FUNCTION_BLOCK DiaglogsContext EXTENDS TcoCore.TcoContext
VAR
    _invokeDiaglog1 : BOOL;
    _dialog1        : TcoCore.TcoDialog(THIS^);
    _dialog2        : TcoCore.TcoDialog(THIS^);
    _dialog3        : TcoCore.TcoDialog(THIS^);
	_dialog4        : TcoCore.TcoDialog(THIS^);

    _invokeDiaglogsConsequential : BOOL;
    _dialog1Consequential        : TcoCore.TcoDialog(THIS^);
    _dialog2Consequential        : TcoCore.TcoDialog(THIS^);
    _dialog3Consequential        : TcoCore.TcoDialog(THIS^);
	
	diag: ITcoDialogAnswer;
	_tonDisposeDialog: TON;
    _state : INT;
	
	
    _invokeCustomizedDiaglog : BOOL;
    _dialogCustomized        : TcoCore.TcoCustomizedDialog(THIS^);
    
END_VAR

(*~
	<docu>
		<summary>
			Main method of the TcoContext. This is the entry point of any control logic that belongs to this context. 
			The call of this method is ensured by calling the <c>InstanceName.Run()</c> method, and it must not be called explicitly.
			This method is abstract, and it must be overridden in derived block.
		</summary>
	</docu>
~*)
METHOD PROTECTED  Main
VAR

END_VAR

CASE _state OF
    0:
        IF (_invokeDiaglog1) THEN
            _state := 10;
		ELSIF (_invokeCustomizedDiaglog) THEN
            _state := 50;
        
        END_IF;
    10:
        _dialog1.Show()
            .WithType(eDialogType.Question)
            .WithYesNoCancel()
			.WithImage('D:\MTS\Develop\TcOpenGroup\TcOpen\assets\logo\TcOpenLogo.png',500,500)
            .WithCaption('Hey 1')
            .WithText('Do we go ahead to 2?');

        IF (_dialog1.Answer = TcoCore.eDialogAnswer.Yes) THEN
            _state := 15;
        END_IF;

        IF (_dialog1.Answer = TcoCore.eDialogAnswer.No) THEN
            _state := 1000;
        END_IF;

        IF (_dialog1.Answer = TcoCore.eDialogAnswer.Cancel) THEN
            _state := 0;
            _invokeDiaglog1 := FALSE;
        END_IF;
    15:
        _dialog1.Show()
            .WithType(eDialogType.Question)
            .WithYesNoCancel()
			.WithImage('',500,500)
            .WithCaption('Hey 2')
            .WithText('Do we go ahead?');

        IF (_dialog1.Answer = TcoCore.eDialogAnswer.Yes) THEN
            _state := 20;
        END_IF;

        IF (_dialog1.Answer = TcoCore.eDialogAnswer.No) THEN
            _state := 1000;
        END_IF;

        IF (_dialog1.Answer = TcoCore.eDialogAnswer.Cancel) THEN
            _state := 0;
            _invokeDiaglog1 := FALSE;
        END_IF;
    20:
        IF (_dialog2.Show()
            .WithType(eDialogType.Info)
            .WithOk()
            .WithCaption('Hey')
            .WithText('We go ahead.')
            .Answer =
            TcoCore.eDialogAnswer.OK) THEN
            _state := 30;
        END_IF
    30:
        _state := 40;
        _tonDisposeDialog(In := FALSE);
    40:
        _tonDisposeDialog(IN := TRUE, PT := T#4S);
		_dialog4.ShowWithExternalClose(inOkAnswerSignal:=FALSE , inYesAnswerSignal:= _tonDisposeDialog.Q, inNoAnswerSignal:= FALSE, inCancelAnswerSignal:= FALSE)
		    .WithType(eDialogType.Info)
            .WithYesNoCancel()
            .WithCaption('Hey')
            .WithText('Do you wana retry it? Yes answer will be set in 4 sec?');

        IF (_dialog4.Answer = TcoCore.eDialogAnswer.Yes) THEN
            _state := 0;
        END_IF;

        IF (_dialog4.Answer = TcoCore.eDialogAnswer.No) THEN
            _state := 50;
        END_IF;

        IF (_dialog4.Answer = TcoCore.eDialogAnswer.Cancel) THEN
            _state := 0;
            _invokeDiaglog1 := FALSE;
        END_IF;
	50:
         _dialogCustomized.Show()
            .WithType(eDialogType.Info)
            .WithOption1('This is Option1=>retry')
			  .WithOption2('This is Option2=>first step')
			    .WithOption3('This is Option3 =>continue')
				  .WithOption4('This is Option4=>stop sequence')
            .WithCaption('Hey')
            .WithText('What we are going to do.');
            
			 IF (_dialogCustomized.Answer = TcoCore.eCustomizedDialogAnswer.Option1) THEN
				_state := 50;
			END_IF;
	
			IF (_dialogCustomized.Answer = TcoCore.eCustomizedDialogAnswer.Option2) THEN
				_state := 0;
			END_IF;
	
			IF (_dialogCustomized.Answer = TcoCore.eCustomizedDialogAnswer.Option3) THEN
				_state := 51;
			END_IF;
	
			IF (_dialogCustomized.Answer = TcoCore.eCustomizedDialogAnswer.Option4) THEN
				_state := 0;
				_invokeCustomizedDiaglog := FALSE;
				_invokeDiaglog1 := FALSE;
			END_IF;
	51:
         _dialogCustomized.Show()
            
            .WithOption1('This is Option1=>retry')
			  .WithOption2('This is Option2=>first step')
			    .WithOption3('This is Option3 =>continue')
			.WithImage('D:\MTS\Develop\TcOpenGroup\TcOpen\assets\logo\TcOpenWide.png',500,500)
            .WithCaption('Hey')
            .WithText('What we are going to do.');
            
			 IF (_dialogCustomized.Answer = TcoCore.eCustomizedDialogAnswer.Option1) THEN
				_state := 50;
			END_IF;
	
			IF (_dialogCustomized.Answer = TcoCore.eCustomizedDialogAnswer.Option2) THEN
				_state := 0;
			END_IF;
	
			IF (_dialogCustomized.Answer = TcoCore.eCustomizedDialogAnswer.Option3) THEN
				_state := 60;
			END_IF;
	
			IF (_dialogCustomized.Answer = TcoCore.eCustomizedDialogAnswer.Option4) THEN
				_state := 0;
				_invokeCustomizedDiaglog := FALSE;
				_invokeDiaglog1 := FALSE;
			END_IF;
     
     
    60:
        _state := 70;
        _tonDisposeDialog(In := FALSE);
	70:
        _tonDisposeDialog(IN := TRUE, PT := T#4S);
		_dialog4.ShowWithExternalClose(inOkAnswerSignal:=FALSE , inYesAnswerSignal:= _tonDisposeDialog.Q, inNoAnswerSignal:= FALSE, inCancelAnswerSignal:= FALSE)
		    .WithType(eDialogType.Info)
            .WithYesNoCancel()
            .WithCaption('Hey')
            .WithText('Do you wana retry it? Yes answer will be set in 4 sec?');

        IF (_dialog4.Answer = TcoCore.eDialogAnswer.Yes) THEN
            _state := 0;
        END_IF;

        IF (_dialog4.Answer = TcoCore.eDialogAnswer.No) THEN
            _state := 80;
        END_IF;

        IF (_dialog4.Answer = TcoCore.eDialogAnswer.Cancel) THEN
            _state := 0;
            _invokeDiaglog1 := FALSE;
        END_IF;
		
	 80:
        _state := 90;
        _tonDisposeDialog(In := FALSE);
	90:
        _tonDisposeDialog(IN := TRUE, PT := T#4S);
		 _dialogCustomized.ShowWithExternalClose(inOption1AnswerSignal:=FALSE,inOption2AnswerSignal:=FALSE, inOption3AnswerSignal:=_tonDisposeDialog.Q,inOption4AnswerSignal:=FALSE)
            
            .WithOption1('This is Option1=>retry')
			  .WithOption2('This is Option2=>first step')
			    .WithOption3('This is Option3 =>continue and finish in 4s')
			.WithImage('D:\MTS\Develop\TcOpenGroup\TcOpen\assets\logo\TcOpenWide.png',500,500)
            .WithCaption('Hey')
            .WithText('What we are going to do.');
            
		
            
			 IF (_dialogCustomized.Answer = TcoCore.eCustomizedDialogAnswer.Option1) THEN
				_state := 80;
			END_IF;
	
			IF (_dialogCustomized.Answer = TcoCore.eCustomizedDialogAnswer.Option2) THEN
				_state := 0;
			END_IF;
	
			IF (_dialogCustomized.Answer = TcoCore.eCustomizedDialogAnswer.Option3) THEN
				_state := 0;
				_invokeCustomizedDiaglog := FALSE;
				_invokeDiaglog1 := FALSE;
			END_IF;
		
	
    1000:
        IF (_dialog3.Show()
            .WithType(eDialogType.Warning)
            .WithOk()
            .WithCaption('Hey')
            .WithText('We don`t go ahead.')
            .Answer =
            TcoCore.eDialogAnswer.OK) THEN
            _state := 0;
        END_IF
END_CASE

//IF(_invokeDiaglog1) THEN

//	IF(_dialog1.Answer = TcoCore.eDialogAnswer.Yes) THEN
//		IF(_dialog2.Show()
//			.WithType(eDialogType.Info)
//			.WithOk()
//			.WithCaption('Hey')
//			.WithText('We go ahead.')
//			.Answer = TcoCore.eDialogAnswer.OK) THEN
//			_invokeDiaglog1 := FALSE;
//		END_IF
//	ELSIF(_dialog1.Answer = TcoCore.eDialogAnswer.No) THEN
//		IF(_dialog3.Show()
//				  	.WithOk()
//					.WithCaption('Hey')
//					.WithText('We don`t go ahead.')
//					.Answer = TcoCore.eDialogAnswer.OK) THEN
//			_invokeDiaglog1 := FALSE;
//		END_IF
//	END_IF			
//END_IF;	

IF (_invokeDiaglogsConsequential) THEN
    _dialog1Consequential.Show().WithYesNoCancel().WithCaption('Hey D1').WithText('D1');
    _dialog2Consequential.Show().WithYesNoCancel().WithCaption('Hey D2').WithText('D2');
    _dialog3Consequential.Show().WithYesNoCancel().WithCaption('Hey D3').WithText('D3');
END_IF;
END_METHOD

END_FUNCTION_BLOCK

(* stored: Version 1.1.0.1
   POU DiaglogsContext: Id {2177bf19-3e21-07f9-0795-125a88ec3524}, SpecialFunc None
   Method Main: Id {e7316bfc-71e9-02be-0fac-515246b2a0e2} *)
